// POUs/CurrentMode/FB_SetCurrentMust
FUNCTION_BLOCK FB_SetCurrentMust
(*************************************************************************************************************************************
**	maxon motor ag
**	elektronik & systemtechnik
**	all rights reserved
**************************************************************************************************************************************
**	Summary :		Write Current Demand Value
**
**	Remarks : 		
**	
**	Created under :	TwinCAT V 2.9.0 (Build 514)
**************************************************************************************************************************************
**	History : 
**	13.10.2003 	| 	san		Beta Version 0.10
**
*************************************************************************************************************************************)
VAR_INPUT
	ADSNetId		: STRING; 	(* Adresses the FC5101 or other Beckhoff CANOpen Masters.
								Can be empty if only local single channel card is present  *)
	NodeId			: INT;		(* Represents the node adress witch is found on Dip Switch of Device *)
	Write			: BOOL;		(* a rising edge starts writing *)

	CurrentMust		: INT;		(* Demand Value *)
END_VAR
VAR_OUTPUT
	Done			: BOOL;		(* Done Flag is set when Function has done *)
	Err				: BOOL;		(* Err Flag is TRUE if an Error has accured, see Errno for more Details *)
	ErrNo			: UDINT;		(* Contains detailed Error Information *)
END_VAR
VAR
	iStep			: INT;
	WriteObj			: ADSWRITE;
	Multiplexor		: UDINT;		(* Gives Index and Subindex of actual Object *)
END_VAR

CASE iStep OF

1:	(* Init *)
	Write := FALSE;
	Done := FALSE;
	Err := FALSE;
	ErrNo := 0;
	WriteObj(WRITE := FALSE);
	iStep := 100;

100:	(* Write Object *)
	WriteObj(
		NETID := ADSNetId,
		PORT := 16#1000 + NodeId,
		IDXGRP := 16#2030,
		IDXOFFS := 0,
		LEN := 2,
		SRCADDR := ADR(CurrentMust),
		WRITE := TRUE,
		TMOUT := t#100ms);
	iStep := 101;
101:  WriteObj();
	IF NOT WriteObj.Busy THEN
		iStep := 102 ;
	END_IF
102:	IF WriteObj.Err THEN
		iStep := 0;
		ErrNo := WriteObj.ErrId;
		Multiplexor := 16#203000;
		Err := TRUE;
	ELSE
		iStep := 0;
	END_IF;
	Done := TRUE;

ELSE
	IF Write THEN
		iStep := 1;
		Done := FALSE;
	END_IF;
END_CASE;

END_FUNCTION_BLOCK

// POUs/Configuration/FB_SetCurrentRegulatorGain
FUNCTION_BLOCK FB_SetCurrentRegulatorGain
(*************************************************************************************************************************************
**	maxon motor ag
**	elektronik & systemtechnik
**	all rights reserved
**************************************************************************************************************************************
**	Summary :		Set Current Regulator Gains (PI)
**
**	Remarks : 		
**
**	Created under :	TwinCAT V 2.9.0 (Build 514)
**************************************************************************************************************************************
**	History : 
**	13.10.2003 	| 	san		Beta Version 0.10
**
*************************************************************************************************************************************)
VAR_INPUT
	ADSNetId		: STRING; 	(* Adresses the FC5101 or other Beckhoff CANOpen Masters.
								Can be empty if only local single channel card is present  *)
	NodeId			: INT;		(* Represents the node adress witch is found on Dip Switch of Device *)

	Write			: BOOL;		(* a rising edge starts writing *)

	P				: UINT;		(* Regulator P - Gain *)
	I				: UINT;		(* Regulator I - Gain  *)
END_VAR
VAR_OUTPUT
	Done			: BOOL;		(* Done Flag is set when Function has done *)
	Err				: BOOL;		(* Err Flag is TRUE if an Error has accured, see Errno for more Details *)
	ErrNo			: UDINT;		(* Contains detailed Error Information *)
END_VAR
VAR
	iStep			: INT;
	WriteP			: ADSWRITE;
	WriteI			: ADSWRITE;
	Multiplexor		: UDINT;		(* Gives Index and Subindex of actual Object *)
END_VAR

CASE iStep OF

1:	(* Init *)
	Write := FALSE;
	Done := FALSE;
	Err := FALSE;
	ErrNo := 0;
	WriteP(WRITE := FALSE);
	WriteI(WRITE := FALSE);
	iStep := 100;

100:	(* Write P - Gain *)
	WriteP(
		NETID := ADSNetId,
		PORT := 16#1000 + NodeId,
		IDXGRP := 16#60F6,
		IDXOFFS := 1,
		LEN := 2,
		SRCADDR := ADR(P),
		WRITE := TRUE,
		TMOUT := t#100ms);
	iStep := 101;
101:  WriteP();
	IF NOT WriteP.Busy THEN
		iStep := 102 ;
	END_IF
102:	IF WriteP.Err THEN
		iStep := 0;
		ErrNo := WriteP.ErrId;
		Multiplexor := 16#60F601;
		Err := TRUE;
	ELSE
		iStep := 200;
	END_IF

200:	(* Write I - Gain *)
	WriteI(
		NETID := ADSNetId,
		PORT := 16#1000 + NodeId,
		IDXGRP := 16#60F6,
		IDXOFFS := 2,
		LEN := 2,
		SRCADDR := ADR(I),
		WRITE := TRUE,
		TMOUT := t#100ms);
	iStep := 201;

201:  WriteI();
	IF NOT WriteI.Busy THEN
		iStep := 202 ;
	END_IF
202:	IF WriteI.Err THEN
		iStep := 0;
		ErrNo := WriteI.ErrId;
		Multiplexor := 16#60F602;
		Err := TRUE;
	ELSE
		iStep := 0;
	END_IF;
	Done := TRUE;

ELSE
	IF Write THEN
		iStep := 1;
		Done := FALSE;
	END_IF;
END_CASE;

END_FUNCTION_BLOCK

// POUs/StateMachine/FB_SetDisableState
FUNCTION_BLOCK FB_SetDisableState
(*************************************************************************************************************************************
**	maxon motor ag
**	elektronik & systemtechnik
**	all rights reserved
**************************************************************************************************************************************
**	Summary :		Disable Device
**
**	Remarks : 	
**
**	Created under :	TwinCAT V 2.9.0 (Build 514)
**************************************************************************************************************************************
**	History : 
**	13.10.2003 	| 	san		Beta Version 0.10
**
*************************************************************************************************************************************)
VAR_INPUT
	ADSNetId		: STRING; 	(* Adresses the FC5101 or other Beckhoff CANOpen Masters.
								Can be empty if only local single channel card is present  *)
	NodeId			: INT;		(* Represents the node adress witch is found on Dip Switch of Device *)
	Write			: BOOL;		(* a rising edge starts writing *)

END_VAR
VAR_OUTPUT

	Done			: BOOL;		(* Done Flag is set when Function has done *)
	Err				: BOOL;		(* Err Flag is TRUE if an Error has accured, see Errno for more Details *)
	ErrNo			: UDINT;		(* Contains detailed Error Information *)
END_VAR
VAR
	iStep			: INT;
	WriteObj			: ADSWRITE;
	Controlword		: UINT	:= 16#0000;
	Multiplexor		: UDINT;		(* Gives Index and Subindex of actual Object *)
END_VAR

CASE iStep OF

1:	(* Init *)
	Write := FALSE;
	Done := FALSE;
	Err := FALSE;
	ErrNo := 0;
	WriteObj(WRITE := FALSE);
	iStep := 100;

100:	(* Write Controlword *)
	WriteObj(
		NETID := ADSNetId,
		PORT := 16#1000 + NodeId,
		IDXGRP := 16#6040,
		IDXOFFS := 0,
		LEN := 2,
		SRCADDR := ADR(Controlword),
		WRITE := TRUE,
		TMOUT := t#100ms);
	iStep := 101;
101:  WriteObj();
	IF NOT WriteObj.Busy THEN
		iStep := 102 ;
	END_IF
102:	IF WriteObj.Err THEN
		iStep := 0;
		ErrNo := WriteObj.ErrId;
		Multiplexor := 16#604000;
		Err := TRUE;
	ELSE
		iStep := 0;
	END_IF;
	Done := TRUE;

ELSE
	IF Write THEN
		iStep := 1;
		Done := FALSE;
	END_IF;
END_CASE;

END_FUNCTION_BLOCK

// POUs/StateMachine/FB_SetEnableState
FUNCTION_BLOCK FB_SetEnableState
(*************************************************************************************************************************************
**	maxon motor ag
**	elektronik & systemtechnik
**	all rights reserved
**************************************************************************************************************************************
**	Summary :		Enable Device
**
**	Remarks : 	
**
**	Created under :	TwinCAT V 2.9.0 (Build 514)
**************************************************************************************************************************************
**	History : 
**	13.10.2003 	| 	san		Beta Version 0.10
**	27.01.2004	|	san		Shutdown only if Status = Switch On Disabled
**
*************************************************************************************************************************************)
VAR_INPUT
	ADSNetId		: STRING; 	(* Adresses the FC5101 or other Beckhoff CANOpen Masters.
								Can be empty if only local single channel card is present  *)
	NodeId			: INT;		(* Represents the node adress witch is found on Dip Switch of Device *)
	Write			: BOOL;		(* a rising edge starts writing *)

END_VAR
VAR_OUTPUT

	Done			: BOOL;		(* Done Flag is set when Function has done *)
	Err				: BOOL;		(* Err Flag is TRUE if an Error has accured, see Errno for more Details *)
	ErrNo			: UDINT;		(* Contains detailed Error Information *)
END_VAR
VAR
	iStep			: INT;
	WriteObj			: ADSWRITE;
	ReadObj			: ADSREAD;
	Controlword		: UINT;
	Statusword		: UINT;		(* Device State *)
	Multiplexor		: UDINT;		(* Gives Index and Subindex of actual Object *)
END_VAR

VAR CONSTANT
	cSwitchOnDisabled		:UINT := 16#0040;
END_VAR

CASE iStep OF

1:	(* Init *)
	Write := FALSE;
	Done := FALSE;
	Err := FALSE;
	ErrNo := 0;
	WriteObj(WRITE := FALSE);
	ReadObj(READ := FALSE);
	iStep := 100;

100:	(* Read Status *)
	ReadObj(
		NETID := ADSNetId,
		PORT := 16#1000 + NodeId,
		IDXGRP := 16#6041,
		IDXOFFS := 0,
		LEN := 2,
		DESTADDR := ADR(Statusword),
		READ := TRUE,
		TMOUT := t#100ms);
	iStep := 101;
101:  ReadObj();
	IF NOT ReadObj.Busy THEN
		iStep := 102 ;
	END_IF
102:	IF ReadObj.Err THEN
		iStep := 0;
		ErrNo := ReadObj.ErrId;
		Multiplexor := 16#604100;
		Err := TRUE;
	ELSE
		IF((UINT_TO_WORD(Statusword) AND 16#006F)  = cSwitchOnDisabled) THEN
			iStep := 200;
		ELSE
			iStep := 300;
		END_IF;
	END_IF;

200:	(* Write Controlword *)
	Controlword := 16#0006; (* Shutdown *)
	WriteObj(
		NETID := ADSNetId,
		PORT := 16#1000 + NodeId,
		IDXGRP := 16#6040,
		IDXOFFS := 0,
		LEN := 2,
		SRCADDR := ADR(Controlword),
		WRITE := TRUE,
		TMOUT := t#100ms);
	iStep := 201;
201:  WriteObj();
	IF NOT WriteObj.Busy THEN
		iStep := 202 ;
	END_IF
202:	IF WriteObj.Err THEN
		iStep := 0;
		ErrNo := WriteObj.ErrId;
		Multiplexor := 16#604000;
		Err := TRUE;
	ELSE
		WriteObj(WRITE := FALSE);
		iStep := 300;
	END_IF;

300:	(* Write Controlword *)
	Controlword := 16#000F; (* Enable Operation *)
	WriteObj(
		NETID := ADSNetId,
		PORT := 16#1000 + NodeId,
		IDXGRP := 16#6040,
		IDXOFFS := 0,
		LEN := 2,
		SRCADDR := ADR(Controlword),
		WRITE := TRUE,
		TMOUT := t#100ms);
	iStep := 301;
301:  WriteObj();
	IF NOT WriteObj.Busy THEN
		iStep := 302 ;
	END_IF
302:	IF WriteObj.Err THEN
		iStep := 0;
		ErrNo := WriteObj.ErrId;
		Multiplexor := 16#604000;
		Err := TRUE;
	ELSE
		iStep := 0;
	END_IF;
	Done := TRUE;

ELSE
	IF Write THEN
		iStep := 1;
		Done := FALSE;
	END_IF;
END_CASE;

END_FUNCTION_BLOCK

// POUs/Configuration/FB_SetEncoderParameter
FUNCTION_BLOCK FB_SetEncoderParameter
(*************************************************************************************************************************************
**	maxon motor ag
**	elektronik & systemtechnik
**	all rights reserved
**************************************************************************************************************************************
**	Summary :		Set Encoder Parameter
**
**	Remarks : 		
**
**	Created under :	TwinCAT V 2.9.0 (Build 514)
**************************************************************************************************************************************
**	History :
**	13.10.2003 	| 	san		Beta Version 0.10
**	21.11.2003	|	san		Beta Version 0.20 firmware changes new SensorType
**
*************************************************************************************************************************************)
VAR_INPUT
	ADSNetId		: STRING; 	(* Adresses the FC5101 or other Beckhoff CANOpen Masters.
								Can be empty if only local single channel card is present  *)
	NodeId			: INT;		(* Represents the node adress witch is found on Dip Switch of Device *)

	Write			: BOOL;		(* a rising edge starts writing *)


	Counts			: UINT;		(* Increments of Incremental Encoder *)
	SensorType		: UINT;		(* Sensor Type*)
END_VAR
VAR_OUTPUT
	Done			: BOOL;		(* Done Flag is set when Function has done *)
	Err				: BOOL;		(* Err Flag is TRUE if an Error has accured, see Errno for more Details *)
	ErrNo			: UDINT;		(* Contains detailed Error Information *)
END_VAR
VAR
	iStep			: INT;
	WriteInc			: ADSWRITE;
	WriteSt			: ADSWRITE;
	Multiplexor		: UDINT;		(* Gives Index and Subindex of actual Object *)
END_VAR

CASE iStep OF

1:	(* Init *)
	Write := FALSE;
	Done := FALSE;
	Err := FALSE;
	ErrNo := 0;
	WriteInc(WRITE := FALSE);
	WriteInc(WRITE := FALSE);
	iStep := 100;

100:	(* Write Encoder Increments *)
	WriteInc(
		NETID := ADSNetId,
		PORT := 16#1000 + NodeId,
		IDXGRP := 16#2210,
		IDXOFFS := 1,
		LEN := 2,
		SRCADDR := ADR(Counts),
		WRITE := TRUE,
		TMOUT := t#100ms);
	iStep := 101;

101:  WriteInc();
	IF NOT WriteInc.Busy THEN
		iStep := 102 ;
	END_IF
102:	IF WriteInc.Err THEN
		iStep := 0;
		ErrNo := WriteInc.ErrId;
		Multiplexor := 16#221001;
		Err := TRUE;
	ELSE
		iStep := 200;
	END_IF

200:	(* Write Sensor Type *)
	WriteSt(
		NETID := ADSNetId,
		PORT := 16#1000 + NodeId,
		IDXGRP := 16#2210,
		IDXOFFS := 2,
		LEN := 2,
		SRCADDR := ADR(SensorType),
		WRITE := TRUE,
		TMOUT := t#100ms);
	iStep := 201;

201:  WriteSt();
	IF NOT WriteSt.Busy THEN
		iStep := 202 ;
	END_IF
202:	IF WriteSt.Err THEN
		iStep := 0;
		ErrNo := WriteSt.ErrId;
		Multiplexor := 16#221002;
		Err := TRUE;
	ELSE
		iStep := 0;
	END_IF
	Done := TRUE;

ELSE
	IF Write THEN
		iStep := 1;
		Done := FALSE;
	END_IF;
END_CASE;

END_FUNCTION_BLOCK

// POUs/HomingMode/FB_SetHomingParameter
FUNCTION_BLOCK FB_SetHomingParameter
(*************************************************************************************************************************************
**	maxon motor ag
**	elektronik & systemtechnik
**	all rights reserved
**************************************************************************************************************************************
**	Summary :		Set all Homing Parameter
**
**	Remarks : 	
**
**	Created under :	TwinCAT V 2.9.0 (Build 514)
**************************************************************************************************************************************
**	History : 
**	30.09.2003 	| 	san		Beta Version 0.10
**	04.02.2004	|	san		CurrentTreshold renamed with CurrentThreshold
**
*************************************************************************************************************************************)
VAR_INPUT
	ADSNetId			: STRING; 	(* Adresses the FC5101 or other Beckhoff CANOpen Masters.
								Can be empty if only local single channel card is present  *)
	NodeId				: INT;		(* Represents the node adress witch is found on Dip Switch of Device *)
	Write				: BOOL;		(* a rising edge starts writing *)

	HomingAcceleration	: UDINT;
	SpeedSwitch			: UDINT;
	SpeedIndex			: UDINT;
	HomeOffset			: DINT;
	CurrentThreshold		: UINT;
END_VAR
VAR_OUTPUT

	Done				: BOOL;		(* Done Flag is set when Function has done *)
	Err					: BOOL;		(* Err Flag is TRUE if an Error has accured, see Errno for more Details *)
	ErrNo				: UDINT;		(* Contains detailed Error Information *)
END_VAR
VAR
	iStep				: INT;
	WriteHomingMethod	: ADSWRITE;
	WriteHomingAcc		: ADSWRITE;
	WriteHomingSpeed	: ADSWRITE;
	WriteSpeedIndex		: ADSWRITE;
	WriteHomeOffset		: ADSWRITE;
	WriteCurTreshold		: ADSWRITE;
	Controlword			: UINT;
	Multiplexor			: UDINT;		(* Gives Index and Subindex of actual Object *)
END_VAR

VAR CONSTANT
	(* HomingMethod *)
	cNegativeLimitSwitch						: SINT := 17;
	cPositiveLimitSwitch						: SINT := 18;
	cHomeSwitchPositiveSpeed				: SINT := 23;
	cHomeSwitchNegativeSpeed				: SINT := 27;
	cCurrentThresholdPositiveSpeed			: SINT := -3;
	cCurrentThresholdNegativeSpeed			: SINT := -4;
	cIndexPositiveSpeed						: SINT := 34;
	cIndexNegativeSpeed						: SINT := 33;
	cNegativeLimitSwitchAndIndex				: SINT := 1;
	cPositiveLimitSwitchAndIndex				: SINT := 2;
	cHomeSwitchPositiveSpeedAndIndex		: SINT := 7;
	cHomeSwitchNegativeSpeedAndIndex		: SINT := 11;
	cCurrentThresholdPositiveSpeedAndIndex	: SINT := -1;
	cCurrentThresholdNegativeSpeedAndIndex	: SINT := -2;
	cActualPosition							: SINT := 35;

END_VAR

CASE iStep OF

1:	(* Init *)
	Write := FALSE;
	Done := FALSE;
	Err := FALSE;
	ErrNo := 0;
	WriteHomingMethod(WRITE := FALSE);
	WriteHomingAcc(WRITE := FALSE);
	WriteHomingSpeed(WRITE := FALSE);
	WriteHomeOffset(WRITE := FALSE);
	WriteCurTreshold(WRITE := FALSE);
	iStep := 100;

100:	(* Write  Speed Index *)
	WriteSpeedIndex(
		NETID := ADSNetId,
		PORT := 16#1000 + NodeId,
		IDXGRP := 16#6099,
		IDXOFFS := 2,
		LEN := 4,
		SRCADDR := ADR(SpeedIndex),
		WRITE := TRUE,
		TMOUT := t#100ms);
	iStep := 101;
101:  WriteSpeedIndex();
	IF NOT WriteSpeedIndex.Busy THEN
		iStep := 102 ;
	END_IF
102:	IF WriteSpeedIndex.Err THEN
		iStep := 0;
		ErrNo := WriteSpeedIndex.ErrId;
		Multiplexor := 16#609902;
		Err := TRUE;
	ELSE
		iStep := 200;
	END_IF

200:	(* Write  Homing Acceleration *)
	WriteHomingAcc(
		NETID := ADSNetId,
		PORT := 16#1000 + NodeId,
		IDXGRP := 16#609A,
		IDXOFFS := 0,
		LEN := 4,
		SRCADDR := ADR(HomingAcceleration),
		WRITE := TRUE,
		TMOUT := t#100ms);
	iStep := 201;
201:  WriteHomingAcc();
	IF NOT WriteHomingAcc.Busy THEN
		iStep := 202 ;
	END_IF
202:	IF WriteHomingAcc.Err THEN
		iStep := 0;
		ErrNo := WriteHomingAcc.ErrId;
		Multiplexor := 16#609A00;
		Err := TRUE;
	ELSE
		iStep := 300;
	END_IF

300:	(* Write  Homing Speed *)
	WriteHomingSpeed(
		NETID := ADSNetId,
		PORT := 16#1000 + NodeId,
		IDXGRP := 16#6099,
		IDXOFFS := 1,
		LEN := 4,
		SRCADDR := ADR(SpeedSwitch),
		WRITE := TRUE,
		TMOUT := t#100ms);
	iStep := 301;
301:  WriteHomingSpeed();
	IF NOT WriteHomingSpeed.Busy THEN
		iStep := 302 ;
	END_IF
302:	IF WriteHomingSpeed.Err THEN
		iStep := 0;
		ErrNo := WriteHomingSpeed.ErrId;
		Multiplexor := 16#609900;
		Err := TRUE;
	ELSE
		iStep := 400;
	END_IF

400:	(* Write  Homing Offset *)
	WriteHomeOffset(
		NETID := ADSNetId,
		PORT := 16#1000 + NodeId,
		IDXGRP := 16#607C,
		IDXOFFS := 0,
		LEN := 4,
		SRCADDR := ADR(HomeOffset),
		WRITE := TRUE,
		TMOUT := t#100ms);
	iStep := 401;
401:  WriteHomeOffset();
	IF NOT WriteHomeOffset.Busy THEN
		iStep := 402 ;
	END_IF
402:	IF WriteHomeOffset.Err THEN
		iStep := 0;
		ErrNo := WriteHomeOffset.ErrId;
		Multiplexor := 16#607C00;
		Err := TRUE;
	ELSE
		iStep := 500;
	END_IF

500:	(* Write  Current Treshold *)
	WriteCurTreshold(
		NETID := ADSNetId,
		PORT := 16#1000 + NodeId,
		IDXGRP := 16#2080,
		IDXOFFS := 0,
		LEN := 2,
		SRCADDR := ADR(CurrentThreshold),
		WRITE := TRUE,
		TMOUT := t#100ms);
	iStep := 501;
501:  WriteCurTreshold();
	IF NOT WriteCurTreshold.Busy THEN
		iStep := 502 ;
	END_IF
502:	IF WriteCurTreshold.Err THEN
		iStep := 0;
		ErrNo := WriteCurTreshold.ErrId;
		Multiplexor := 16#208000;
		Err := TRUE;
	ELSE
		iStep := 0;
	END_IF
	Done := TRUE;

ELSE
	IF Write THEN
		iStep := 1;
		Done := FALSE;
	END_IF;
END_CASE;

END_FUNCTION_BLOCK

// POUs/Configuration/FB_SetMotorParameter
FUNCTION_BLOCK FB_SetMotorParameter
(*************************************************************************************************************************************
**	maxon motor ag
**	elektronik & systemtechnik
**	all rights reserved
**************************************************************************************************************************************
**	Summary :		Set Motor Parameters
**
**	Remarks : 		
**
**	Created under :	TwinCAT V 2.9.0 (Build 514)
**************************************************************************************************************************************
**	History : 
**	13.10.2003 	| 	san		Beta Version 0.10
**	21.11.2003	|	san		Beta Version 0.20 firmware changes in object 6410
**
*************************************************************************************************************************************)
VAR_INPUT
	ADSNetId		: STRING; 	(* Adresses the FC5101 or other Beckhoff CANOpen Masters.
								Can be empty if only local single channel card is present  *)
	NodeId			: INT;		(* Represents the node adress witch is found on Dip Switch of Device *)

	Write			: BOOL;		(* a rising edge starts writing *)

	MotorType			: INT;		(*    10: Ec Motor	(Brushless Motor)
										1: Dc Motor	(Brushed Motor) *)

	ContinuousCurrent		: UINT;		(* Continuous Current *)
	PeakCurrent			: UINT;		(* Peak Current (normaly 2 * Icont) *)
	PolePair				: USINT;		(* Motor Pole Pair  *)
	ThermalTimeConstant	: UINT;		(* Thermal Time Constant *)
END_VAR
VAR_OUTPUT
	Done			: BOOL;		(* Done Flag is set when Function has done *)
	Err				: BOOL;		(* Err Flag is TRUE if an Error has accured, see Errno for more Details *)
	ErrNo			: UDINT;		(* Contains detailed Error Information *)
END_VAR
VAR
	iStep			: INT;
	WriteMTyp		: ADSWRITE;
	WriteKm			: ADSWRITE;
	WriteIcont		: ADSWRITE;
	WriteIpeak		: ADSWRITE;
	WritePolePair		: ADSWRITE;
	WriteTt			: ADSWRITE;
	Multiplexor		: UDINT;		(* Gives Index and Subindex of actual Object *)
END_VAR

CASE iStep OF

1:	(* Init *)
	Write := FALSE;
	Done := FALSE;
	Err := FALSE;
	ErrNo := 0;
	WriteMTyp(WRITE := FALSE);
	WriteKm(WRITE := FALSE);
	WriteIcont(WRITE := FALSE);
	WriteIpeak(WRITE := FALSE);
	WritePolePair(WRITE := FALSE);
	WriteTt(WRITE := FALSE);
	iStep := 100;

100:	(* Set Motor Type *)
	WriteMTyp(
		NETID := ADSNetId,
		PORT := 16#1000 + NodeId,
		IDXGRP := 16#6402,
		IDXOFFS := 0,
		LEN := 2,
		SRCADDR := ADR(MotorType),
		WRITE := TRUE,
		TMOUT := t#100ms);
	iStep := 101;
101:  WriteMTyp();
	IF NOT WriteMTyp.Busy THEN
		iStep := 102 ;
	END_IF
102:	IF WriteMTyp.Err THEN
		iStep := 0;
		ErrNo := WriteMTyp.ErrId;
		Multiplexor := 16#640200;
		Err := TRUE;
	ELSE
		iStep := 200;
	END_IF

200:	(* Set Continuous Current *)
	WriteKm(
		NETID := ADSNetId,
		PORT := 16#1000 + NodeId,
		IDXGRP := 16#6410,
		IDXOFFS := 1,
		LEN := 2,
		SRCADDR := ADR(ContinuousCurrent),
		WRITE := TRUE,
		TMOUT := t#100ms);
	iStep := 201;
201:  WriteKm();
	IF NOT WriteKm.Busy THEN
		iStep := 202 ;
	END_IF
202:	IF WriteKm.Err THEN
		iStep := 0;
		ErrNo := WriteKm.ErrId;
		Multiplexor := 16#641001;
		Err := TRUE;
	ELSE
		iStep := 300;
	END_IF

300:	(* Set Peak Current *)
	WriteIcont(
		NETID := ADSNetId,
		PORT := 16#1000 + NodeId,
		IDXGRP := 16#6410,
		IDXOFFS := 2,
		LEN := 2,
		SRCADDR := ADR(PeakCurrent),
		WRITE := TRUE,
		TMOUT := t#100ms);
	iStep := 301;
301:  WriteIcont();
	IF NOT WriteIcont.Busy THEN
		iStep := 302 ;
	END_IF
302:	IF WriteIcont.Err THEN
		iStep := 0;
		ErrNo := WriteIcont.ErrId;
		Multiplexor := 16#641002;
		Err := TRUE;
	ELSE
		iStep := 400;
	END_IF

400:	(* Set Number of Pole Pair *)
	IF (PolePair = 0) THEN
		iStep := 500;
	ELSE
		WritePolePair(
			NETID := ADSNetId,
			PORT := 16#1000 + NodeId,
			IDXGRP := 16#6410,
			IDXOFFS := 3,
			LEN := 1,
			SRCADDR := ADR(PolePair),
			WRITE := TRUE,
			TMOUT := t#100ms);
		iStep := 401;
	END_IF;
401:  WritePolePair();
	IF NOT WritePolePair.Busy THEN
		iStep := 402 ;
	END_IF
402:	IF WritePolePair.Err THEN
		iStep := 0;
		ErrNo := WritePolePair.ErrId;
		Multiplexor := 16#641003;
		Err := TRUE;
	ELSE
		iStep := 500;
	END_IF

500:	(* Set Thermal Time Constant*)
	WriteTt(
		NETID := ADSNetId,
		PORT := 16#1000 + NodeId,
		IDXGRP := 16#6410,
		IDXOFFS := 5,
		LEN := 2,
		SRCADDR := ADR(ThermalTimeConstant),
		WRITE := TRUE,
		TMOUT := t#100ms);
	iStep := 501;
501:  WriteTt();
	IF NOT WriteTt.Busy THEN
		iStep := 502 ;
	END_IF
502:	IF WriteTt.Err THEN
		iStep := 0;
		ErrNo := WriteTt.ErrId;
		Multiplexor := 16#641006;
		Err := TRUE;
	ELSE
		iStep := 0;
	END_IF;
	Done := TRUE;

ELSE
	IF Write THEN
		iStep := 1;
		Done:= FALSE;
	END_IF;
END_CASE;

END_FUNCTION_BLOCK

// POUs/Utilities/FB_SetObject
FUNCTION_BLOCK FB_SetObject
(*************************************************************************************************************************************
**	maxon motor ag
**	elektronik & systemtechnik
**	all rights reserved
**************************************************************************************************************************************
**	Summary :		writes one object from object dictionary
**
**	Remarks : 	
**
**	Created under :	TwinCAT V 2.9.0 (Build 514)
**************************************************************************************************************************************
**	History : 
**	13.10.2003 	| 	san		Beta Version 0.10
**	04.02.2004	|	san		ODIdx renamed witth ObjectIndex, ODSubidx renamed with ObjectSubindex
**
*************************************************************************************************************************************)
VAR_INPUT
	ADSNetId		: STRING; 	(* Adresses the FC5101 or other Beckhoff CANOpen Masters.
								Can be empty if only local single channel card is present  *)
	NodeId			: INT;		(* Represents the node adress witch is found on Dip Switch of Device *)
	Write			: BOOL;		(* a rising edge starts writing *)

	ObjectIndex		: UINT;		(* Object Dictionary Index *)
	ObjectSubindex	: USINT;		(* Object Dictionary Sub Index *)
	Len				: USINT;		(* Length of Object, Number of Bytes *)
	Data			: UDINT;		(* Data to be written *)

END_VAR
VAR_OUTPUT
	Done			: BOOL;		(* Done Flag is set when Function has done *)
	Err				: BOOL;		(* Err Flag is TRUE if an Error has accured, see Errno for more Details *)
	ErrNo			: UDINT;		(* Contains detailed Error Information *)
END_VAR
VAR
	iStep			: INT;
	WriteObj			: ADSWRITE;
	Multiplexor		: UDINT;		(* Gives Index and Subindex of actual Object *)
END_VAR

CASE iStep OF

1:	(* Init *)
	Write := FALSE;
	Done := FALSE;
	Err := FALSE;
	ErrNo := 0;
	WriteObj(WRITE := FALSE);
	iStep := 100;

100:	(* Write Object *)
	WriteObj(
		NETID := ADSNetId,
		PORT := 16#1000 + NodeId,
		IDXGRP := ObjectIndex,
		IDXOFFS := ObjectSubindex,
		LEN := LEN,
		SRCADDR := ADR(Data),
		WRITE := TRUE,
		TMOUT := t#100ms);
	iStep := 101;
101:  WriteObj();
	IF NOT WriteObj.Busy THEN
		iStep := 102 ;
	END_IF
102:	IF WriteObj.Err THEN
		iStep := 0;
		ErrNo := WriteObj.ErrId;
		Multiplexor := ObjectIndex * 256; (* Shift of 8 *)
		Multiplexor := Multiplexor + ObjectSubindex;
		Err := TRUE;
	ELSE
		iStep := 0;
	END_IF;
	Done := TRUE;

ELSE
	IF Write THEN
		iStep := 1;
		Done := FALSE;
	END_IF;
END_CASE;

END_FUNCTION_BLOCK

// POUs/StateMachine/FB_SetOperationMode
FUNCTION_BLOCK FB_SetOperationMode
(*************************************************************************************************************************************
**	maxon motor ag
**	elektronik & systemtechnik
**	all rights reserved
**************************************************************************************************************************************
**	Summary :		Set Operation Mode
**
**	Remarks : 	
**
**	Created under :	TwinCAT V 2.9.0 (Build 514)
**************************************************************************************************************************************
**	History : 
**	13.10.2003 	| 	san		Beta Version 0.10
**	04.02.2004	|	san		type of Mode changed from USINT to SINT
**
*************************************************************************************************************************************)
VAR_INPUT
	ADSNetId		: STRING; 	(* Adresses the FC5101 or other Beckhoff CANOpen Masters.
								Can be empty if only local single channel card is present  *)
	NodeId			: INT;		(* Represents the node adress witch is found on Dip Switch of Device *)
	Write			: BOOL;		(* a rising edge starts writing *)

	Mode			: SINT;		(* Operation Mode:
									16#01	= 	ProfilePositonMode
									16#03	= 	ProfileVelocityMode
									16#06	= 	HomingMode
									16#FF	= 	PositonMode
									16#FE	= 	VelocityMode
									16#FD	= 	CurrentMode
									 *)
END_VAR
VAR_OUTPUT

	Done			: BOOL;		(* Done Flag is set when Function has done *)
	Err				: BOOL;		(* Err Flag is TRUE if an Error has accured, see Errno for more Details *)
	ErrNo			: UDINT;		(* Contains detailed Error Information *)
END_VAR
VAR
	iStep			: INT;
	WriteObj			: ADSWRITE;
	Multiplexor		: UDINT;		(* Gives Index and Subindex of actual Object *)
END_VAR

CASE iStep OF

1:	(* Init *)
	Write := FALSE;
	Done := FALSE;
	Err := FALSE;
	ErrNo := 0;
	WriteObj(WRITE := FALSE);
	iStep := 100;

100:	(* Write Mode *)
	WriteObj(
		NETID := ADSNetId,
		PORT := 16#1000 + NodeId,
		IDXGRP := 16#6060,
		IDXOFFS := 0,
		LEN := 1,
		SRCADDR := ADR(Mode),
		WRITE := TRUE,
		TMOUT := t#100ms);
	iStep := 101;
101:  WriteObj();
	IF NOT WriteObj.Busy THEN
		iStep := 102 ;
	END_IF
102:	IF WriteObj.Err THEN
		iStep := 0;
		ErrNo := WriteObj.ErrId;
		Multiplexor := 16#606000;
		Err := TRUE;
	ELSE
		iStep := 0;
	END_IF
	Done := TRUE;

ELSE
	IF Write THEN
		iStep := 1;
		Done := FALSE;
	END_IF;
END_CASE;

END_FUNCTION_BLOCK

// POUs/PositionMode/FB_SetPositionMust
FUNCTION_BLOCK FB_SetPositionMust
(*************************************************************************************************************************************
**	maxon motor ag
**	elektronik & systemtechnik
**	all rights reserved
**************************************************************************************************************************************
**	Summary :		Write Position Demand Value
**
**	Remarks : 		
**
**	Created under:	TwinCAT V 2.9.0 (Build 514)
**************************************************************************************************************************************
**	History : 
**	13.10.2003 	| 	san		Beta Version 0.10
**
*************************************************************************************************************************************)
VAR_INPUT
	ADSNetId		: STRING; 	(* Adresses the FC5101 or other Beckhoff CANOpen Masters.
								Can be empty if only local single channel card is present  *)
	DevAddr			: INT;		(* Adresses the maxon Device (Example: EPOS).
								Represents the node adress witch is found on Dip Switch of Device *)
	Write			: BOOL;		(* a rising edge starts writing *)

	PositionMust		: DINT;		(* Demand Value *)

END_VAR
VAR_OUTPUT

	Done			: BOOL;		(* Done Flag is set when Function has done *)
	Err				: BOOL;		(* Err Flag is TRUE if an Error has accured, see Errno for more Details *)
	ErrNo			: UDINT;		(* Contains detailed Error Information *)
END_VAR
VAR
	iStep			: INT;
	WriteObj			: ADSWRITE;
	Multiplexor		: UDINT;		(* Gives Index and Subindex of actual Object *)
END_VAR

CASE iStep OF

1:	(* Init *)
	Write := FALSE;
	Done := FALSE;
	Err := FALSE;
	ErrNo := 0;
	WriteObj(WRITE := FALSE);
	iStep := 100;

100:	(* Write Object *)
	WriteObj(
		NETID := ADSNetId,
		PORT := 16#1000 + DevAddr,
		IDXGRP := 16#2062,
		IDXOFFS := 0,
		LEN := 4,
		SRCADDR := ADR(PositionMust),
		WRITE := TRUE,
		TMOUT := t#100ms);
	iStep := 101;
101:  WriteObj();
	IF NOT WriteObj.Busy THEN
		iStep := 102 ;
	END_IF
102:	IF WriteObj.Err THEN
		iStep := 0;
		ErrNo := WriteObj.ErrId;
		Multiplexor := 16#206200;
		Err := TRUE;
	ELSE
		iStep := 0;
	END_IF;
	Done := TRUE;

ELSE
	IF Write THEN
		iStep := 1;
		Done := FALSE;
	END_IF;
END_CASE;

END_FUNCTION_BLOCK

// POUs/ProfilePositionMode/FB_SetPositionProfile
FUNCTION_BLOCK FB_SetPositionProfile
(*************************************************************************************************************************************
**	maxon motor ag
**	elektronik & systemtechnik
**	all rights reserved
**************************************************************************************************************************************
**	Summary :		Set Position Profile
**
**	Remarks : 		
**
**	Created under:	TwinCAT V 2.9.0 (Build 514)
**************************************************************************************************************************************
**	History : 
**	13.10.2003 	| 	san		Beta Version 0.10
**
*************************************************************************************************************************************)
VAR_INPUT
	ADSNetId		: STRING; 	(* Adresses the FC5101 or other Beckhoff CANOpen Masters.
								Can be empty if only local single channel card is present  *)
	NodeId			: INT;		(*Represents the node adress witch is found on Dip Switch of Device *)

	Write			: BOOL;		(* a rising edge starts writing *)

	ProfileVelocity	: UDINT;		(* Profile Velocity *)
	ProfileAcceleration: UDINT;		(* Profile Acceleration *)
	ProfileDeceleration: UDINT;		(* Profile Deceleration *)
END_VAR
VAR_OUTPUT
	Done			: BOOL;		(* Done Flag is set when Function has done *)
	Err				: BOOL;		(* Err Flag is TRUE if an Error has accured, see Errno for more Details *)
	ErrNo			: UDINT;		(* Contains detailed Error Information *)
END_VAR
VAR
	iStep			: INT;
	WriteVel			: ADSWRITE;
	WriteAcc			: ADSWRITE;
	WriteDec		: ADSWRITE;
	Multiplexor		: UDINT;		(* Gives Index and Subindex of actual Object *)
END_VAR

CASE iStep OF

1:	(* Init *)
	Write := FALSE;
	Done := FALSE;
	Err := FALSE;
	ErrNo := 0;
	WriteVel(WRITE := FALSE);
	WriteAcc(WRITE := FALSE);
	WriteDec(WRITE := FALSE);
	iStep := 100;

100:	(* Profile Velocity *)
	WriteVel(
		NETID := ADSNetId,
		PORT := 16#1000 + NodeId,
		IDXGRP := 16#6081,
		IDXOFFS := 0,
		LEN := 4,
		SRCADDR := ADR(ProfileVelocity),
		WRITE := TRUE,
		TMOUT := t#100ms);
	iStep := 101;
101:  WriteVel ();
	IF NOT WriteVel.Busy THEN
		iStep := 102 ;
	END_IF
102:	IF WriteVel.Err THEN
		iStep := 0;
		ErrNo := WriteVel.ErrId;
		Multiplexor := 16#608100;
		Err := TRUE;
	ELSE
		iStep := 200;
	END_IF

200:	(* Profile Acceleration *)
	WriteAcc(
		NETID := ADSNetId,
		PORT := 16#1000 + NodeId,
		IDXGRP := 16#6083,
		IDXOFFS := 0,
		LEN := 4,
		SRCADDR := ADR(ProfileAcceleration),
		WRITE := TRUE,
		TMOUT := t#100ms);
	iStep := 201;
201:  WriteAcc ();
	IF NOT WriteAcc.Busy THEN
		iStep := 202 ;
	END_IF
202:	IF WriteAcc.Err THEN
		iStep := 0;
		ErrNo := WriteAcc.ErrId;
		Multiplexor := 16#608300;
		Err := TRUE;
	ELSE
		iStep := 300;
	END_IF

300:	(* Profile Deceleration *)
	WriteDec(
		NETID := ADSNetId,
		PORT := 16#1000 + NodeId,
		IDXGRP := 16#6084,
		IDXOFFS := 0,
		LEN := 4,
		SRCADDR := ADR(ProfileDeceleration),
		WRITE := TRUE,
		TMOUT := t#100ms);
	iStep := 301;
301:  WriteDec ();
	IF NOT WriteDec.Busy THEN
		iStep := 302 ;
	END_IF
302:	IF WriteDec.Err THEN
		iStep := 0;
		ErrNo := WriteDec.ErrId;
		Multiplexor := 16#608400;
		Err := TRUE;
	ELSE
		iStep := 0;
	END_IF
	Done := TRUE;

ELSE
	IF Write THEN
		iStep := 1;
		Done := FALSE ;
	END_IF;
END_CASE;

END_FUNCTION_BLOCK

// POUs/Configuration/FB_SetPositionRegulatorGain
FUNCTION_BLOCK FB_SetPositionRegulatorGain
(*************************************************************************************************************************************
**	maxon motor ag
**	elektronik & systemtechnik
**	all rights reserved
**************************************************************************************************************************************
**	Summary :		Set Position Regulator Gains (PID)
**
**	Remarks : 		
**
**	Created under :	TwinCAT V 2.9.0 (Build 514)
**************************************************************************************************************************************
**	History : 
**	13.10.2003 	| 	san		Beta Version 0.10
**
*************************************************************************************************************************************)
VAR_INPUT
	ADSNetId		: STRING; 	(* Adresses the FC5101 or other Beckhoff CANOpen Masters.
								Can be empty if only local single channel card is present  *)
	NodeId			: INT;		(* Represents the node adress witch is found on Dip Switch of Device *)

	Write			: BOOL;		(* a rising edge starts writing *)

	P				: UINT;		(* Position Regulator P - Gain *)
	I				: UINT;		(* Position Regulator I - Gain  *)
	D				: UINT;		(* Position Regulator D - Gain *)
END_VAR
VAR_OUTPUT
	Done			: BOOL;		(* Done Flag is set when Function has done *)
	Err				: BOOL;		(* Err Flag is TRUE if an Error has accured, see Errno for more Details *)
	ErrNo			: UDINT;		(* Contains detailed Error Information *)
END_VAR
VAR
	iStep			: INT;
	WriteP			: ADSWRITE;
	WriteI			: ADSWRITE;
	WriteD			: ADSWRITE;
	Multiplexor		: UDINT;		(* Gives Index and Subindex of actual Object *)
END_VAR

CASE iStep OF

1:	(* Init *)
	Write := FALSE;
	Done := FALSE;
	Err := FALSE;
	ErrNo := 0;
	WriteP(WRITE := FALSE);
	WriteI(WRITE := FALSE);
	WriteD(WRITE := FALSE);
	iStep := 100;

100:	(* Write P - Gain *)
	WriteP(
		NETID := ADSNetId,
		PORT := 16#1000 + NodeId,
		IDXGRP := 16#60FB,
		IDXOFFS := 1,
		LEN := 2,
		SRCADDR := ADR(P),
		WRITE := TRUE,
		TMOUT := t#100ms);
	iStep := 101;
101:  WriteP();
	IF NOT WriteP.Busy THEN
		iStep := 102 ;
	END_IF
102:	IF WriteP.Err THEN
		iStep := 0;
		ErrNo := WriteP.ErrId;
		Multiplexor := 16#60FB01;
		Err := TRUE;
	ELSE
		iStep := 200;
	END_IF

200:	(* Write I - Gain *)
	WriteI(
		NETID := ADSNetId,
		PORT := 16#1000 + NodeId,
		IDXGRP := 16#60FB,
		IDXOFFS := 2,
		LEN := 2,
		SRCADDR := ADR(I),
		WRITE := TRUE,
		TMOUT := t#100ms);
	iStep := 201;
201:  WriteI();
	IF NOT WriteI.Busy THEN
		iStep := 202 ;
	END_IF
202:	IF WriteI.Err THEN
		iStep := 0;
		ErrNo := WriteI.ErrId;
		Multiplexor := 16#60FB02;
		Err := TRUE;
	ELSE
		iStep := 300;
	END_IF

300:	(* Write D - Gain *)
	WriteD(
		NETID := ADSNetId,
		PORT := 16#1000 + NodeId,
		IDXGRP := 16#60FB,
		IDXOFFS := 3,
		LEN := 2,
		SRCADDR := ADR(D),
		WRITE := TRUE,
		TMOUT := t#100ms);
	iStep := 301;
301:  WriteD();
	IF NOT WriteD.Busy THEN
		iStep := 302 ;
	END_IF
302:	IF WriteD.Err THEN
		iStep := 0;
		ErrNo := WriteD.ErrId;
		Multiplexor := 16#60FB03;
		Err := TRUE;
	ELSE
		iStep := 0;
	END_IF;
	Done := TRUE;

ELSE
	IF Write THEN
		iStep := 1;
		Done := FALSE;
	END_IF;
END_CASE;

END_FUNCTION_BLOCK

// POUs/StateMachine/FB_SetQuickStopState
FUNCTION_BLOCK FB_SetQuickStopState
(*************************************************************************************************************************************
**	maxon motor ag
**	elektronik & systemtechnik
**	all rights reserved
**************************************************************************************************************************************
**	Summary :		Quick Stop Device
**
**	Remarks : 	
**
**	Created under :	TwinCAT V 2.9.0 (Build 514)
**************************************************************************************************************************************
**	History : 
**	13.10.2003 	| 	san		Beta Version 0.10
**
*************************************************************************************************************************************)
VAR_INPUT
	ADSNetId		: STRING; 	(* Adresses the FC5101 or other Beckhoff CANOpen Masters.
								Can be empty if only local single channel card is present  *)
	NodeId			: INT;		(* Represents the node adress witch is found on Dip Switch of Device *)
	Write			: BOOL;		(* a rising edge starts writing *)

END_VAR
VAR_OUTPUT

	Done			: BOOL;		(* Done Flag is set when Function has done *)
	Err				: BOOL;		(* Err Flag is TRUE if an Error has accured, see Errno for more Details *)
	ErrNo			: UDINT;		(* Contains detailed Error Information *)
END_VAR
VAR
	iStep			: INT;
	WriteObj			: ADSWRITE;
	Controlword		: UINT	:= 16#0002;
	Multiplexor		: UDINT;		(* Gives Index and Subindex of actual Object *)
END_VAR

CASE iStep OF

1:	(* Init *)
	Write := FALSE;
	Done := FALSE;
	Err := FALSE;
	ErrNo := 0;
	WriteObj(WRITE := FALSE);
	iStep := 100;

100:	(* Write Controlword *)
	WriteObj(
		NETID := ADSNetId,
		PORT := 16#1000 + NodeId,
		IDXGRP := 16#6040,
		IDXOFFS := 0,
		LEN := 2,
		SRCADDR := ADR(Controlword),
		WRITE := TRUE,
		TMOUT := t#100ms);
	iStep := 101;
101:  WriteObj();
	IF NOT WriteObj.Busy THEN
		iStep := 102 ;
	END_IF
102:	IF WriteObj.Err THEN
		iStep := 0;
		ErrNo := WriteObj.ErrId;
		Multiplexor := 16#604000;
		Err := TRUE;
	ELSE
		iStep := 0;
	END_IF;
	Done := TRUE;

ELSE
	IF Write THEN
		iStep := 1;
		Done := FALSE;
	END_IF;
END_CASE;

END_FUNCTION_BLOCK

// POUs/VelocityMode/FB_SetVelocityMust
FUNCTION_BLOCK FB_SetVelocityMust
(*************************************************************************************************************************************
**	maxon motor ag
**	elektronik & systemtechnik
**	all rights reserved
**************************************************************************************************************************************
**	Summary :		Write Velocity Demand Value
**
**	Remarks : 		
**
**	Created under:	TwinCAT V 2.9.0 (Build 514)
**************************************************************************************************************************************
**	History : 
**	13.10.2003 	| 	san		Beta Version 0.10
**
*************************************************************************************************************************************)
VAR_INPUT
	ADSNetId		: STRING; 	(* Adresses the FC5101 or other Beckhoff CANOpen Masters.
								Can be empty if only local single channel card is present  *)
	NodeId			: INT;		(* Represents the node adress witch is found on Dip Switch of Device *)
	Write			: BOOL;		(* a rising edge starts writing *)

	VelocityMust		: DINT;		(* Demand Value *)

END_VAR
VAR_OUTPUT
	Done			: BOOL;		(* Done Flag is set when Function has done *)
	Err				: BOOL;		(* Err Flag is TRUE if an Error has accured, see Errno for more Details *)
	ErrNo			: UDINT;		(* Contains detailed Error Information *)
END_VAR
VAR
	iStep			: INT;
	WriteObj			: ADSWRITE;
	Multiplexor		: UDINT;		(* Gives Index and Subindex of actual Object *)
END_VAR

CASE iStep OF

1:	(* Init *)
	Write := FALSE;
	Done := FALSE;
	Err := FALSE;
	ErrNo := 0;
	WriteObj(WRITE := FALSE);
	iStep := 100;

100:	(* Write Object *)
	WriteObj(
		NETID := ADSNetId,
		PORT := 16#1000 + NodeId,
		IDXGRP := 16#206B,
		IDXOFFS := 0,
		LEN := 4,
		SRCADDR := ADR(VelocityMust),
		WRITE := TRUE,
		TMOUT := t#100ms);
	iStep := 101;
101:  WriteObj();
	IF NOT WriteObj.Busy THEN
		iStep := 102 ;
	END_IF
102:	IF WriteObj.Err THEN
		iStep := 0;
		ErrNo := WriteObj.ErrId;
		Multiplexor := 16#206B00;
		Err := TRUE;
	ELSE
		iStep := 0;
	END_IF;
	Done := TRUE;

ELSE
	IF Write THEN
		iStep := 1;
		Done := FALSE;
	END_IF;
END_CASE;

END_FUNCTION_BLOCK

// POUs/ProfileVelocityMode/FB_SetVelocityProfile
FUNCTION_BLOCK FB_SetVelocityProfile
(*************************************************************************************************************************************
**	maxon motor ag
**	elektronik & systemtechnik
**	all rights reserved
**************************************************************************************************************************************
**	Summary :		Set Velocity Profile
**
**	Remarks : 		
**
**	Created under:	TwinCAT V 2.9.0 (Build 514)
**************************************************************************************************************************************
**	History : 
**	13.10.2003 	| 	san		Beta Version 0.10
**
*************************************************************************************************************************************)
VAR_INPUT
	ADSNetId		: STRING; 	(* Adresses the FC5101 or other Beckhoff CANOpen Masters.
								Can be empty if only local single channel card is present  *)
	NodeId			: INT;		(* Represents the node adress witch is found on Dip Switch of Device *)
	Write			: BOOL;		(* a rising edge starts writing *)

	ProfileAcceleration: UDINT;		(* Profile Acceleration *)
	ProfileDeceleration: UDINT;		(* Profile Deceleration *)
END_VAR
VAR_OUTPUT
	Done			: BOOL;		(* Done Flag is set when Function has done *)
	Err				: BOOL;		(* Err Flag is TRUE if an Error has accured, see Errno for more Details *)
	ErrNo			: UDINT;		(* Contains detailed Error Information *)
END_VAR
VAR
	iStep			: INT;
	WriteAcc			: ADSWRITE;
	WriteDec		: ADSWRITE;
	Multiplexor		: UDINT;		(* Gives Index and Subindex of actual Object *)
END_VAR

CASE iStep OF

1:	(* Init *)
	Write := FALSE;
	Done := FALSE;
	Err := FALSE;
	ErrNo := 0;
	WriteAcc(WRITE := FALSE);
	WriteDec(WRITE := FALSE);
	iStep := 100;

100:	(* Profile Acceleration *)
	WriteAcc(
		NETID := ADSNetId,
		PORT := 16#1000 + NodeId,
		IDXGRP := 16#6083,
		IDXOFFS := 0,
		LEN := 4,
		SRCADDR := ADR(ProfileAcceleration),
		WRITE := TRUE,
		TMOUT := t#100ms);
	iStep := 101;
101:  WriteAcc();
	IF NOT WriteAcc.Busy THEN
		iStep := 102 ;
	END_IF
102:	IF WriteAcc.Err THEN
		iStep := 0;
		ErrNo := WriteAcc.ErrId;
		Multiplexor := 16#608300;
		Err := TRUE;
	ELSE
		iStep := 200;
	END_IF

200:	(* Profile Deceleration *)
	WriteDec(
		NETID := ADSNetId,
		PORT := 16#1000 + NodeId,
		IDXGRP := 16#6084,
		IDXOFFS := 0,
		LEN := 4,
		SRCADDR := ADR(ProfileDeceleration),
		WRITE := TRUE,
		TMOUT := t#100ms);
	iStep := 201;
201:  WriteDec();
	IF NOT WriteDec.Busy THEN
		iStep := 202 ;
	END_IF
202:	IF WriteDec.Err THEN
		iStep := 0;
		ErrNo := WriteDec.ErrId;
		Multiplexor := 16#608400;
		Err := TRUE;
	ELSE
		iStep := 0;
	END_IF
	Done := TRUE;

ELSE
	IF Write THEN
		iStep := 1;
		Done := FALSE;
	END_IF;
END_CASE;

END_FUNCTION_BLOCK

// POUs/Configuration/FB_SetVelocityRegulatorGain
FUNCTION_BLOCK FB_SetVelocityRegulatorGain
(*************************************************************************************************************************************
**	maxon motor ag
**	elektronik & systemtechnik
**	all rights reserved
**************************************************************************************************************************************
**	Summary :		Set Velocity Regulator Gains (PI)
**
**	Remarks : 		
**
**	Created under :	TwinCAT V 2.9.0 (Build 514)
**************************************************************************************************************************************
**	History : 
**	13.10.2003 	| 	san		Beta Version 0.10
**
*************************************************************************************************************************************)
VAR_INPUT
	ADSNetId		: STRING; 	(* Adresses the FC5101 or other Beckhoff CANOpen Masters.
								Can be empty if only local single channel card is present  *)
	NodeId			: INT;		(* Represents the node adress witch is found on Dip Switch of Device *)
	Write			: BOOL;		(* a rising edge starts writing *)

	P				: UINT;		(* Regulator P - Gain *)
	I				: UINT;		(* Regulator I - Gain  *)
END_VAR
VAR_OUTPUT
	Done			: BOOL;		(* Done Flag is set when Function has done *)
	Err				: BOOL;		(* Err Flag is TRUE if an Error has accured, see Errno for more Details *)
	ErrNo			: UDINT;		(* Contains detailed Error Information *)
END_VAR
VAR
	iStep			: INT;
	WriteP			: ADSWRITE;
	WriteI			: ADSWRITE;
	Multiplexor		: UDINT;		(* Gives Index and Subindex of actual Object *)
END_VAR

CASE iStep OF

1:	(* Init *)
	Write := FALSE;
	Done := FALSE;
	Err := FALSE;
	ErrNo := 0;
	WriteP(WRITE := FALSE);
	WriteI(WRITE := FALSE);
	iStep := 100;

100:	(* Write P - Gain *)
	WriteP(
		NETID := ADSNetId,
		PORT := 16#1000 + NodeId,
		IDXGRP := 16#60F9,
		IDXOFFS := 1,
		LEN := 2,
		SRCADDR := ADR(P),
		WRITE := TRUE,
		TMOUT := t#100ms);
	iStep := 101;
101:  WriteP();
	IF NOT WriteP.Busy THEN
		iStep := 102 ;
	END_IF
102:	IF WriteP.Err THEN
		iStep := 0;
		ErrNo := WriteP.ErrId;
		Multiplexor := 16#60F901;
		Err := TRUE;
	ELSE
		iStep := 200;
	END_IF

200:	(* Write I - Gain *)
	WriteI(
		NETID := ADSNetId,
		PORT := 16#1000 + NodeId,
		IDXGRP := 16#60F9,
		IDXOFFS := 2,
		LEN := 2,
		SRCADDR := ADR(I),
		WRITE := TRUE,
		TMOUT := t#100ms);
	iStep := 201;
201:  WriteI();
	IF NOT WriteI.Busy THEN
		iStep := 202 ;
	END_IF
202:	IF WriteI.Err THEN
		iStep := 0;
		ErrNo := WriteI.ErrId;
		Multiplexor := 16#60F902;
		Err := TRUE;
	ELSE
		iStep := 0;
	END_IF;
	Done := TRUE;

ELSE
	IF Write THEN
		iStep := 1;
		Done := FALSE;
	END_IF;
END_CASE;

END_FUNCTION_BLOCK

// POUs/HomingMode/FB_StopHoming
FUNCTION_BLOCK FB_StopHoming
(*************************************************************************************************************************************
**	maxon motor ag
**	elektronik & systemtechnik
**	all rights reserved
**************************************************************************************************************************************
**	Summary :		Stop Homing
**
**	Remarks : 	
**
**	Created under :	TwinCAT V 2.9.0 (Build 514)
**************************************************************************************************************************************
**	History : 
**	30.09.2003 	| 	san		Beta Version 0.10
**
*************************************************************************************************************************************)
VAR_INPUT
	ADSNetId			: STRING; 	(* Adresses the FC5101 or other Beckhoff CANOpen Masters.
									    Can be empty if only local single channel card is present  *)
	NodeId				: INT;		(* Represents the node adress witch is found on Dip Switch of Device *)
	Write				: BOOL;		(* a rising edge starts writing *)

END_VAR
VAR_OUTPUT

	Done				: BOOL;		(* Done Flag is set when Function has done *)
	Err					: BOOL;		(* Err Flag is TRUE if an Error has accured, see Errno for more Details *)
	ErrNo				: UDINT;		(* Contains detailed Error Information *)
END_VAR
VAR
	iStep				: INT;
	WriteCw				: ADSWRITE;
	Controlword			: UINT;
	Statusword			: UINT;
	Multiplexor			: UDINT;		(* Gives Index and Subindex of actual Object *)
END_VAR

CASE iStep OF

1:	(* Init *)
	Write := FALSE;
	Done := FALSE;
	Err := FALSE;
	ErrNo := 0;
	WriteCw(WRITE := FALSE);
	iStep := 100;

100:	(* Write  Controlword *)
	Controlword := 16#010F;
	WriteCw(
		NETID := ADSNetId,
		PORT := 16#1000 + NodeId,
		IDXGRP := 16#6040,
		IDXOFFS := 0,
		LEN := 2,
		SRCADDR := ADR(Controlword),
		WRITE := TRUE,
		TMOUT := t#100ms);
	iStep := 101;
101:  WriteCw();
	IF NOT WriteCw.Busy THEN
		iStep := 102 ;
	END_IF
102:	IF WriteCw.Err THEN
		iStep := 0;
		ErrNo := WriteCw.ErrId;
		Multiplexor := 16#604000;
		Err := TRUE;
	ELSE
		iStep := 0;
	END_IF
	Done := TRUE;

ELSE
	IF Write THEN
		iStep := 1;
		Done := FALSE;
	END_IF;
END_CASE;

END_FUNCTION_BLOCK

// POUs/Utilities/FB_Store
FUNCTION_BLOCK FB_Store
(*************************************************************************************************************************************
**	maxon motor ag
**	elektronik & systemtechnik
**	all rights reserved
**************************************************************************************************************************************
**	Summary :		store all system parameters
**
**	Remarks : 	
**
**	Created under :	TwinCAT V 2.9.0 (Build 514)
**************************************************************************************************************************************
**	History : 
**	13.10.2003 	| 	san		Beta Version 0.10
**
*************************************************************************************************************************************)
VAR_INPUT
	ADSNetId		: STRING; 	(* Adresses the FC5101 or other Beckhoff CANOpen Masters.
								Can be empty if only local single channel card is present  *)
	NodeId			: INT;		(* Represents the node adress witch is found on Dip Switch of Device *)
	Write			: BOOL;		(* a rising edge starts writing *)

END_VAR
VAR_OUTPUT
	Done			: BOOL;		(* Done Flag is set when Function has done *)
	Err				: BOOL;		(* Err Flag is TRUE if an Error has accured, see Errno for more Details *)
	ErrNo			: UDINT;		(* Contains detailed Error Information *)
END_VAR
VAR
	iStep			: INT;
	WriteObj			: ADSWRITE;
	udiData: 			UDINT			:= 16#65766173;
	Multiplexor		: UDINT;		(* Gives Index and Subindex of actual Object *)
END_VAR

CASE iStep OF

1:	(* Init *)
	Write := FALSE;
	Done := FALSE;
	Err := FALSE;
	ErrNo := 0;
	WriteObj(WRITE := FALSE);
	iStep := 100;

100:	(* Read Object *)
	WriteObj(
		NETID := ADSNetId,
		PORT := 16#1000 + NodeId,
		IDXGRP := 16#1010,
		IDXOFFS := 1,
		LEN := 4,
		SRCADDR := ADR(udiData),
		WRITE := TRUE,
		TMOUT := t#100ms);
	iStep := 101;
101:  WriteObj();
	IF NOT WriteObj.Busy THEN
		iStep := 102 ;
	END_IF
102:	IF WriteObj.Err THEN
		iStep := 0;
		ErrNo := WriteObj.ErrId;
		Multiplexor := 16#101001;
		Err := TRUE;
	ELSE
		iStep := 0;
	END_IF;
	Done := TRUE;

ELSE
	IF Write THEN
		iStep := 1;
		Done := FALSE;
	END_IF;
END_CASE;

END_FUNCTION_BLOCK
